Universal Robots PolyScope program: step0_register_echo_500hz.urp

Program step0_register_echo_500hz (installation=default directory=/programs/andyl/kunwei createdIn=5.11.9.1010452 lastSavedIn=5.11.9.1010452 robotSerialNumber=20225200364)
Calibrated DH parameters: a=[0.00002, -0.569483, -0.54992, -0.00001, -0.000036, 0]; d=[0.180894, -146.691669, 192.918669, -46.053088, 0.119778, 0.115602]; alpha=[1.571425, -0.001534, 0.003359, 1.568739, -1.571477, 0]; deltaTheta=[0, 0.376258, -0.101074, -0.275185, -0.000002, 0]
Robot Program (runOnlyOnce=true)
  Script file /programs/andyl/kunwei/step0_register_echo_500hz.script
    | # Step0 high-rate 500 Hz Kunwei RTDE input-register echo, no motion.
    | # VERSION: 2026-06-05T1741HKT_500HZ_ECHO_V2
    | # GENERATED_AT_LOCAL: 2026-06-05T17:41:33+0800
    | # Run from a PolyScope Script node only after the Python step0 bridge/benchmark
    | # is writing input_double_register_24..36. This program only mirrors values to
    | # output_double_register_24..35 for the Ubuntu logger.
    | 
    | def codex_step0_register_echo():
    |   textmsg("codex step0 500hz register echo version 2026-06-05T1741HKT_500HZ_ECHO_V2 start")
    |   local t = 0.0
    |   local dt = 0.002
    |   local loop_counter = 0.0
    |   while t < 120.0:
    |     local normal_force = read_input_float_register(24)
    |     local force_norm = read_input_float_register(25)
    |     local heartbeat = read_input_float_register(26)
    |     local sensor_ok = read_input_float_register(27)
    |     local stop_request = read_input_float_register(28)
    |     local target_force = read_input_float_register(29)
    |     local torque_norm = read_input_float_register(30)
    |     local fx = read_input_float_register(31)
    |     local fy = read_input_float_register(32)
    |     local fz = read_input_float_register(33)
    |     local mx = read_input_float_register(34)
    |     local my = read_input_float_register(35)
    |     write_output_float_register(24, normal_force)
    |     write_output_float_register(25, force_norm)
    |     write_output_float_register(26, heartbeat)
    |     write_output_float_register(27, sensor_ok)
    |     write_output_float_register(28, stop_request)
    |     write_output_float_register(29, target_force)
    |     write_output_float_register(30, torque_norm)
    |     write_output_float_register(31, fx)
    |     write_output_float_register(32, fy)
    |     write_output_float_register(33, fz)
    |     write_output_float_register(34, mx)
    |     write_output_float_register(35, loop_counter)
    |     sync()
    |     loop_counter = loop_counter + 1.0
    |     t = t + dt
    |   end
    |   textmsg("codex step0 500hz register echo version 2026-06-05T1741HKT_500HZ_ECHO_V2 done")
    | end
    | 
    | codex_step0_register_echo()
